Fanuc KAREL source: kt00208.KL

-- PROVISIONAL review KL for V940-1; original PC SHA256 513c402e8f3d27a8fb89be5beab801ce04187dce061c44233bdc9163062af1ca
-- Incomplete behavior may be omitted. Consult companion uncertainty JSON. Do not deploy.
PROGRAM KT00208
%NOLOCKGROUP
VAR
  I1 : INTEGER
  OUT : INTEGER
-- UNRESOLVED_DECL H2 type=002017
BEGIN
  -- V9_ZERO_TABLE_METADATA_HINT layout=0001; no indexed target words; source/name/runtime held
  -- UNRESOLVED_PC offsets 5-16; opcodes 2E,23
  -- UNRESOLVED_PC offsets 21-35; opcodes 2E,22,9D,33,B4
  -- UNRESOLVED_PC offsets 40-62; opcodes 21,22,9D,33,B3,46,23
  -- UNRESOLVED_PC offsets 67-71; opcodes 7F
END KT00208
